TYPE "UDT_HMI_Alarm_V2"
VERSION : 0.1
   STRUCT
      t : Struct
         x0 : Bool;
         x1 : Bool;
         x2 : Bool;
         x3 : Bool;
         x4 : Bool;
         x5 : Bool;
         x6 : Bool;
         x7 : Bool;
         x8 : Bool;
         x9 : Bool;
         x10 : Bool;
         x11 : Bool;
         x12 : Bool;
         x13 : Bool;
         x14 : Bool;
         x15 : Bool;
      END_STRUCT;
      iHmiSumAlm : Word;
   END_STRUCT;

END_TYPE

TYPE "UDT_Tilting_Alm"
VERSION : 0.1
   STRUCT
      tEmergencyAlarm { S7_SetPoint := 'False'} : Array["STARTARRAY".."DALARM"] of "UDT_HMI_Alarm_V2";   // stop machine fault
      tAlarm { S7_SetPoint := 'False'} : Array["STARTARRAY".."DALARM"] of "UDT_HMI_Alarm_V2";   // stop next cycle faults
      tWarning { S7_SetPoint := 'False'} : Array["STARTARRAY".."DALARM"] of "UDT_HMI_Alarm_V2";   // Generic warning
   END_STRUCT;

END_TYPE

TYPE "UDT_Tilting_Hmi"
VERSION : 0.1
   STRUCT
      tHMR { ExternalWritable := 'False'} : Struct   // {[Unit]|[Scada Unit]|[LowLimit]|[HigLimit]|[Acces]}
         xForcedUp { ExternalWritable := 'False'} : Bool;   // Main Tiltin Forced Up  {x|x|x|x|O}
         xForcedDw { ExternalWritable := 'False'} : Bool;   // Main Tiltin Forced Dw {x|x|x|x|O}
         xBrakerOK { ExternalWritable := 'False'} : Bool;   // Braker ok
         xAutomatic { ExternalWritable := 'False'} : Bool;   // Main Tiltin Autoamtic {x|x|x|x|O}
         xMaintenanceModeSelector { ExternalWritable := 'False'} : Bool;   // Mainteannce Mode Selctor
         xAllToCulletByButtons { ExternalWritable := 'False'} : Bool;   // All to cullet by Button
         xMaintenanceBarUp { ExternalWritable := 'False'} : Bool;   // Maintenance Bar UP {x|x|x|x|O}
         sDescritionGoDown { ExternalWritable := 'False'} : String;   // Description String
         tManCmd { ExternalWritable := 'False'} : Struct
            xCmdRise { ExternalWritable := 'False'} : Bool;   // Manual Command Rise {x|x|x|x|O}
            xCmdDown { ExternalWritable := 'False'} : Bool;   // Manual Command Descend{x|x|x|x|O}
         END_STRUCT;
      END_STRUCT;
      tHMW : Struct   // {[Unit]|[Scada Unit]|[LowLimit]|[HigLimit]|[Acces]}
         xForceUp : Bool;   // Main Tiltin Force Up  {x|x|x|x|O}
         xForceDw : Bool;   // Main Tiltin Force Dw {x|x|x|x|O}
         xAutomatic : Bool;   // Main Tiltin Force Automatic {x|x|x|x|O}
         tManCmd : Struct
            xCmdRise : Bool;   // Manual Command Rise {x|x|x|x|O}
            xCmdDown : Bool;   // Manual Command Descend{x|x|x|x|O}
         END_STRUCT;
      END_STRUCT;
   END_STRUCT;

END_TYPE

DATA_BLOCK "Tilting_Alm"
{ S7_Optimized_Access := 'FALSE' }
VERSION : 0.1
NON_RETAIN
   STRUCT
      rgtInd { S7_SetPoint := 'False'} : Array["STARTARRAY".."DMAXTILTING"] of "UDT_Tilting_Alm";
   END_STRUCT;


BEGIN

END_DATA_BLOCK

DATA_BLOCK "Tilting_Hmi"
{ S7_Optimized_Access := 'FALSE' }
VERSION : 0.1
NON_RETAIN
   STRUCT
      rgtInd { S7_SetPoint := 'False'} : Array["STARTARRAY".."DMAXTILTING"] of "UDT_Tilting_Hmi";
   END_STRUCT;


BEGIN

END_DATA_BLOCK

